// TwinCAT 3 PLC project TcIotOcppServerDynamicStationsPlc
// Title: TwinCAT IoT OCPP Dynamic Stations Sample
// Company: Beckhoff Automation GmbH & Co. KG
// ProjectVersion: 1.0.0.0
// ProgramVersion: 3.1.4026.10
// libraries:
//   Tc2_Standard, * (Beckhoff Automation GmbH)
//   Tc2_System, * (Beckhoff Automation GmbH)
//   Tc3_Module, * (Beckhoff Automation GmbH)
//   Tc3_OCPP, * (Beckhoff Automation GmbH)
// project tree:
//   DUTs/ ST_StationData.TcDUT
//   GVLs/ VAR_OCPP.TcGVL
//   / PlcTask.TcTTO
//   POUs/ F_AuthStatus.TcPOU, MAIN.TcPOU
// real-time tasks:
//   TASK PlcTask: cycle T#10ms, priority 20, ADS port 350

CONFIGURATION TcIotOcppServerDynamicStationsPlc
    RESOURCE PLC ON TwinCAT3
        TASK PlcTask(INTERVAL := T#10ms, PRIORITY := 20);
        PROGRAM MAIN WITH PlcTask : MAIN;
    END_RESOURCE
END_CONFIGURATION

// ---- DUTs/ST_StationData.TcDUT
TYPE ST_StationData :
STRUCT
	hStationId : UDINT;
	sIdent : T_OCPP_Identity;
	sAuthHash : T_OCPP_Hash;

	// charging station
	bOpen : BOOL;
	nHeartbeats : UDINT;
	eStationStatus : E_OCPP1_ChargePointStatus;
	eConnector1Status : E_OCPP1_ChargePointStatus;
	eConnector2Status : E_OCPP1_ChargePointStatus;
	// boot notification
	sModel : STRING(31); // Required. This contains a value that identifies the model of the ChargePoint.
	sVendor : STRING(31); // Required. This contains a value that identifies the vendor of the ChargePoint.
	sChargeBoxSerial : STRING(31); // Optional. This contains a value that identifies the serial number of the Charge Box inside the Charge Point.
	sChargePointSerial : STRING(31); // Optional. This contains a value that identifies the serial number of the Charge Point.
	sFirmwareVersion : STRING(63); // Optional. This contains the firmware version of the Charge Point.
	sMeterSerial : STRING(31); // Optional. This contains the serial number of the main electrical meter of the Charge Point.
	sMeterType : STRING(31); // Optional. This contains the type of the main electrical meter of the Charge Point.
END_STRUCT
END_TYPE

// ---- GVLs/VAR_OCPP.TcGVL
{attribute 'qualified_only'}
VAR_GLOBAL
	arrStationList : ARRAY[1..nStationListMax] OF ST_StationData := [
		( sIdent := 'Test01', sAuthHash := '083bb79c338a0d6dd768b46ca7a320d56c270e15236e30b4f0007d75bcbeb20e' ),
		( sIdent := 'Test02', sAuthHash := '70bf8db192a798cd72cc3b657627f9e712d96ea615caeea6898f2b5b83793f4f' )
	];
	arrAuthList : ARRAY[1..nAuthListMax] OF ST_OCPP1_AuthorizationData := [
		( sIdTag := 'B45E00EE', stIdTagInfo := ( eStatus := E_OCPP1_AuthorizationStatus.Accepted ) ),
		( sIdTag := 'A46FF2F1', stIdTagInfo := ( eStatus := E_OCPP1_AuthorizationStatus.Accepted ) ),
		( sIdTag := '1234abcd', stIdTagInfo := ( eStatus := E_OCPP1_AuthorizationStatus.Accepted ) )
	];

	stServerParam : ST_OCPP1_ServerParam := (
		//nOID := 16#01010010); // ObjectID of the TcIotOcpp Client Object (0 to create a new instance).
		nTaskOID := 16#02010030, // ObjectId of the Task whose shall execute the client (0 to use I/O Idle Task)
		sHost := '0.0.0.0', // Defines the server-address by host-name, domain-name or IP-address.
		nPort := 8080, // Defines the server-port.
		sPath := 'ocpp', // Defines the server-path.
		eAuthMode := E_OCPP1_AuthenticationMode.None, // Defines an optional authentication-mode.
		//eAuthMode := E_OCPP1_AuthenticationMode.Basic, // Defines an optional authentication-mode.
		eEncryptionMode := E_OCPP_EncryptionMode.None, // Defines an optional encryption mode.
		//eEncryptionMode := E_OCPP_EncryptionMode.Enable, // Defines an optional encryption mode.
		//sCaFile := '%TC_TARGETPATH%\Certificates\CA.crt', // Certificate of the certificate authority (CA) as filename (PEM or DER format).
		//sCrtFile := '%TC_TARGETPATH%\Certificates\OCPP.crt', // Certificate of the server (public key) as filename (PEM or DER format)
		//sKeyFile := '%TC_TARGETPATH%\Certificates\OCPP.key', // Key of the server (private key) as filename (PEM or DER format).
		eTraceLevel := TcTraceLevel.tlVerbose); // Defines the maximum trace level of ADS log messages
END_VAR
VAR_GLOBAL CONSTANT
	nStationListMax : UDINT := 256;
	nAuthListMax : UDINT := 3;
END_VAR

// ---- POUs/MAIN.TcPOU
PROGRAM MAIN
VAR
	bValid : BOOL;
	bInitialized : BOOL;
	fbServer : FB_OCPP1_Server(VAR_OCPP.stServerParam);

	nIdx : UDINT;
	mStationData : REFERENCE TO ST_StationData;
	// receive
	bRecv : BOOL;
	hStationId : UDINT;
	eAction : E_OCPP1_Action;
	hMessageId : T_OCPP_MessageId;
	// status notification
	nStatusConnectorId : UDINT;
	eStatusNotificationError : E_OCPP1_ChargePointError;
	eStatusNotificationStatus : E_OCPP1_ChargePointStatus;
	// transactional
	sIdTag: T_OCPP1_IdToken;
	eAuthStatus : E_OCPP1_AuthorizationStatus;
	nTransactionId : UDINT;
	sDataTransferData : T_OCPP1_DataTransferData;
	arrSampledValues : ARRAY[1..10] OF ST_OCPP1_SampledValue;
END_VAR

bValid := fbServer.bValid;
IF NOT bValid THEN RETURN; END_IF

IF NOT bInitialized THEN
	FOR nIdx := 1 TO VAR_OCPP.nStationListMax DO
		IF VAR_OCPP.arrStationList[nIdx].sIdent <> '' THEN
			fbServer.CreateStation(VAR_OCPP.arrStationList[nIdx].sIdent, VAR_OCPP.arrStationList[nIdx].sAuthHash, hStationId => VAR_OCPP.arrStationList[nIdx].hStationId);
		END_IF
	END_FOR
	bInitialized := TRUE;
END_IF

IF fbServer.PollRequest(hStationId => hStationId, eAction => eAction, hMessageId => hMessageId) THEN
	bRecv := FALSE;
	FOR nIdx := 1 TO VAR_OCPP.nStationListMax DO
		IF VAR_OCPP.arrStationList[nIdx].hStationId = hStationId THEN
			mStationData REF= VAR_OCPP.arrStationList[nIdx];
			bRecv := TRUE;
			EXIT;
		END_IF
	END_FOR
	IF NOT bRecv THEN
		fbServer.RespError(hStationId, hMessageId, eAction, E_OCPP1_Error.GenericError);
	ELSE
		CASE eAction OF
			E_OCPP1_Action.Heartbeat:
				IF fbServer.RecvHeartbeat(hStationId, hMessageId => hMessageId) THEN
					mStationData.nHeartbeats := mStationData.nHeartbeats + 1;
					fbServer.RespHeartbeat(hStationId, hMessageId);
				END_IF

			E_OCPP1_Action.BootNotification:
				IF fbServer.RecvBootNotification(hStationId, hMessageId=> hMessageId,
					sModel=> mStationData.sModel, sVendor=> mStationData.sVendor,
					sChargeBoxSerial=> mStationData.sChargeBoxSerial, sChargePointSerial=> mStationData.sChargePointSerial,
					sFirmwareVersion=> mStationData.sFirmwareVersion, sMeterSerial=> mStationData.sMeterSerial,
					sMeterType=> mStationData.sMeterType)
				THEN
					fbServer.RespBootNotification(hStationId, hMessageId, eStatus := E_OCPP1_RegistrationStatus.Accepted);
				END_IF

			E_OCPP1_Action.MeterValues:
				IF fbServer.RecvMeterValue(hStationId, hMessageId => hMessageId, aSampleValues := arrSampledValues) THEN
					fbServer.RespMeterValue(hStationId, hMessageId);
				END_IF
			E_OCPP1_Action.StatusNotification:
				IF fbServer.RecvStatusNotification(hStationId, hMessageId => hMessageId,
					nConnectorId => nStatusConnectorId, eError => eStatusNotificationError, eStatus => eStatusNotificationStatus)
				THEN
					CASE nStatusConnectorId OF
						0: mStationData.eStationStatus := eStatusNotificationStatus;
						1: mStationData.eConnector1Status := eStatusNotificationStatus;
						2: mStationData.eConnector2Status := eStatusNotificationStatus;
					END_CASE
					fbServer.RespStatusNotification(hStationId, hMessageId);
				END_IF
			E_OCPP1_Action.Authorize:
				IF fbServer.RecvAuthorize(hStationId, hMessageId => hMessageId, sIdTag => sIdTag) THEN
					fbServer.RespAuthorize(hStationId, hMessageId, eStatus := F_AuthStatus(sIdTag));
				END_IF
			E_OCPP1_Action.StartTransaction:
				IF fbServer.RecvStartTransaction(hStationId, hMessageId => hMessageId, sIdTag => sIdTag) THEN
					eAuthStatus := F_AuthStatus(sIdTag);
					IF eAuthStatus = E_OCPP1_AuthorizationStatus.Accepted THEN
						nTransactionId := nTransactionId + 1;
						fbServer.RespStartTransaction(hStationId, hMessageId, eStatus := E_OCPP1_AuthorizationStatus.Accepted, nTransactionId := nTransactionId);
					ELSE
						fbServer.RespStartTransaction(hStationId, hMessageId, eStatus := E_OCPP1_AuthorizationStatus.Invalid, nTransactionId := 0);
					END_IF
				END_IF
			E_OCPP1_Action.StopTransaction:
				IF fbServer.RecvStopTransaction(hStationId, hMessageId => hMessageId, sIdTag => sIdTag) THEN
					eAuthStatus := F_AuthStatus(sIdTag);
					IF eAuthStatus = E_OCPP1_AuthorizationStatus.Accepted THEN
						fbServer.RespStopTransaction(hStationId, hMessageId, eStatus := E_OCPP1_AuthorizationStatus.Accepted);
					ELSE
						fbServer.RespStopTransaction(hStationId, hMessageId, eStatus := E_OCPP1_AuthorizationStatus.Invalid);
					END_IF
				END_IF
			E_OCPP1_Action.DiagnosticsStatusNotification:
				IF fbServer.RecvDiagnosticsStatusNotification(hStationId, hMessageId => hMessageId) THEN
					fbServer.RespDiagnosticsStatusNotification(hStationId, hMessageId);
				END_IF
			E_OCPP1_Action.FirmwareStatusNotification:
				IF fbServer.RecvFirmwareStatusNotification(hStationId, hMessageId => hMessageId) THEN
					fbServer.RespFirmwareStatusNotification(hStationId, hMessageId);
				END_IF
			E_OCPP1_Action.DataTransfer:
				IF fbServer.RecvDataTransfer(hStationId, hMessageId => hMessageId, sData := sDataTransferData) THEN
					fbServer.RespDataTransfer(hStationId, hMessageId, eStatus := E_OCPP1_DataTransferStatus.Accepted);
				END_IF
			E_OCPP1_Action.SecurityEventNotification:
				IF fbServer.RecvSecurityEventNotification(hStationId, hMessageId => hMessageId) THEN
					fbServer.RespSecurityEventNotification(hStationId, hMessageId);
				END_IF
		ELSE
			fbServer.RespError(hStationId, hMessageId, eAction, E_OCPP1_Error.NotImplemented);
		END_CASE
	END_IF
END_IF

END_PROGRAM

// ---- POUs/F_AuthStatus.TcPOU
FUNCTION F_AuthStatus : E_OCPP1_AuthorizationStatus
VAR_IN_OUT
	sIdTag: T_OCPP1_IdToken;
END_VAR
VAR
	nIdx : UDINT;
END_VAR

F_AuthStatus := E_OCPP1_AuthorizationStatus.Invalid;
FOR nIdx := 1 TO VAR_OCPP.nAuthListMax DO
	IF VAR_OCPP.arrAuthList[nIdx].sIdTag = sIdTag THEN
		F_AuthStatus := VAR_OCPP.arrAuthList[nIdx].stIdTagInfo.eStatus;
		RETURN;
	END_IF
END_FOR

END_FUNCTION
